INTERFACE ITF_Tree_IndexBased

METHOD AddNodeAsChildByName : BOOL
VAR_INPUT
    sNewName    : STRING;
    sParentName : STRING;
END_VAR
END_METHOD

END_INTERFACE

(* stored: Version 1.1.0.1, ProductVersion 3.1.4024.11
   Itf ITF_Tree_IndexBased: Id {6c15a641-a3e1-429e-975b-7d04725a2547}
   Method AddNodeAsChildByName: Id {b2e07763-97dd-4243-a177-e38b66773085} *)
